TYPE U_TestOverlay :
UNION
    nRaw : UDINT;
    arrBytes : ARRAY[0..3] OF BYTE;
END_UNION
END_TYPE

(* stored: Version 1.1.0.1
   DUT U_TestOverlay: Id {55555555-5555-5555-5555-555555555504} *)
